INTERFACE I_MotionDriveStateMachine

PROPERTY MoveState : E_MOVESTATE
GET
END_GET
END_PROPERTY

METHOD StateMachine
VAR_INPUT
	InterlockEvent : BOOL;
	Error : BOOL;
END_VAR
END_METHOD

PROPERTY WatchDogStatus : BOOL
GET
END_GET
END_PROPERTY

PROPERTY WatchDogTimeOut : BOOL
GET
END_GET
END_PROPERTY

END_INTERFACE

(* stored: Version 1.1.0.1
   Itf I_MotionDriveStateMachine: Id {40b216ee-9f46-47cd-9746-7ef949a43466}
   Property MoveState: Id {e8643675-62f4-49b4-a123-32f66c1fe60c}
   Get Get: Id {ad4a13f0-51ea-427f-a59a-e1cbc3d762f5}
   Method StateMachine: Id {95486653-d40f-4598-a1e5-f89d76b3879d}
   Property WatchDogStatus: Id {84ab4881-15ff-4eca-a59f-21a36f427ff1}
   Get Get: Id {2e343ed6-211d-437b-8645-05aaaac04a5e}
   Property WatchDogTimeOut: Id {c783fed4-2455-40e1-810c-36b1d1e0a3ec}
   Get Get: Id {1d23ddbf-2686-4e13-8f77-1400bd225647} *)
